TYPE VTD_Shuttle_Interlock_DUT :
STRUCT
	Interlock_Complete:  BOOL;
	Interlock_Complete_Ack:  BOOL;
	Ready_To_Interlock:  Bool;
	Interlock_Request:  Bool;
	Shuttle_ID:  UInt;
	Shuttle_Target_Location:  DInt;
	Shuttle_Start_Location:  DInt;
	Shuttle_Loaded:  Bool;
	Shuttle_Interlock_Task_ID:  UInt;
	Shuttle_Interlock_Task_Metadata:  STRING;
END_STRUCT
END_TYPE

(* stored: Version 1.1.0.1
   DUT VTD_Shuttle_Interlock_DUT: Id {2bb361bb-29f4-4dbe-b279-802fc704d8e0} *)
